{attribute 'GeneratedUsingTerminal: EK1100-0000-0018'}
{attribute addProperty BoxType "EK1100-0000-0018"}
{attribute addProperty Id "Beckhoff_EL66xxEK1122Beckhoff_EL66xxEK1122_DCCAD5BD273A_0001_EL6601_0000_0000EL6601_EEB2FEF410A_0002_EL6601_0000_0001EL6601_EEB2FEF410A_0003_EL6601_0000_0016EL6601_EEB2FEF410A_0004_EL6601_0000_0017EL6601_EEB2FEF410A_0005_EL6601_0000_0018EL6601_EEB2FEF410A_0006_EL6601_0000_0019EL6601_EEB2FEF410A_0007_EL6601_0000_0021EL6601_EEB2FEF410A_0008_EL6614_0000_0016EL6614_EEB2FEF410A_0009_EL6614_0000_0017EL6614_EEB2FEF410A_0010_EL6614_0000_0018EL6614_EEB2FEF410A_0011_EL6614_0000_0019EL6614_EEB2FEF410A_0012_EL6614_0000_0021EL6614_EEB2FEF410A_0013_EL6631_0000_0016EL6631_210A1A8D16A_0014_EL6631_0000_0017EL6631_210A1A8D16A_0015_EL6631_0000_0018EL6631_210A1A8D16A_0016_EL6631_0010_0016EL6631_210A1A8D16A_0017_EL6631_0010_0017EL6631_210A1A8D16A_0018_EL6631_0010_0018EL6631_210A1A8D16A_0019_EL6652_0000_0017EL6652_210A1A8D16A_0020_EL6652_0000_0018EL6652_210A1A8D16A_0021_EL6652_0010_0017EL6652_210A1A8D16A_0022_EL6652_0010_0018EL6652_210A1A8D16A_0023_EL6688_0000_0016EL6688_8DEED67724A_0024_EL6688_0000_0017EL6688_747A9CEE44A_0025_EL6688_0000_0018EL6688_747A9CEE44A_0026_EL6688_0000_0019EL6688_747A9CEE44A_0027_EL6688_0000_0020EL6688_747A9CEE44A_0028_EL6688_0000_0022EL6688_747A9CEE44A_0029_EL6690_0001_0000EL6690_FD149FC213A_0030_EL6690_0001_0016EL6690_FD149FC213A_0031_EL6690_0001_0017EL6690_FD149FC213A_0037_EL6692_0000_0016EL6692_F12D40B324A_0038_EL6692_0000_0017EL6692_F12D40B324A_0039_EL6692_0000_0018EL6692_F12D40B324A_0045_EL6695_0000_0001EL6695_258CDFB421A_0047_EL6695_0000_0002EL6695_258CDFB421A_0049_EL6695_0000_0003EL6695_258CDFB421A_0051_EL6695_0000_0004EL6695_258CDFB421A_0053_EL6695_0000_0005EL6695_258CDFB421A_0055_EL6695_0000_0006EL6695_258CDFB421"}
{attribute addProperty CRC "854866809"}
{attribute addProperty Size "1034"}
TYPE Beckhoff_EL66xx_32F43B79 EXTENDS EK1100_1FC0878B :
STRUCT
	{attribute addProperty Name "Beckhoff EL66xxEK1122"}
	{attribute addProperty PreviousPort "Beckhoff EL66xx : B"}
	Beckhoff_EL66xxEK1122 : Beckhoff_EL66xxEK1122_DCCAD5BD;
	{attribute addProperty Name "A_0001(EL6601-0000-0000)"}
	{attribute addProperty PreviousPort "Beckhoff EL66xxEK1122 : C"}
	A_0001_EL6601_0000_0000 : EL6601_EEB2FEF4;
	{attribute addProperty Name "A_0002(EL6601-0000-0001)"}
	{attribute addProperty PreviousPort "A_0001(EL6601-0000-0000) : B"}
	A_0002_EL6601_0000_0001 : EL6601_EEB2FEF4;
	{attribute addProperty Name "A_0003(EL6601-0000-0016)"}
	{attribute addProperty PreviousPort "A_0002(EL6601-0000-0001) : B"}
	A_0003_EL6601_0000_0016 : EL6601_EEB2FEF4;
	{attribute addProperty Name "A_0004(EL6601-0000-0017)"}
	{attribute addProperty PreviousPort "A_0003(EL6601-0000-0016) : B"}
	A_0004_EL6601_0000_0017 : EL6601_EEB2FEF4;
	{attribute addProperty Name "A_0005(EL6601-0000-0018)"}
	{attribute addProperty PreviousPort "A_0004(EL6601-0000-0017) : B"}
	A_0005_EL6601_0000_0018 : EL6601_EEB2FEF4;
	{attribute addProperty Name "A_0006(EL6601-0000-0019)"}
	{attribute addProperty PreviousPort "A_0005(EL6601-0000-0018) : B"}
	A_0006_EL6601_0000_0019 : EL6601_EEB2FEF4;
	{attribute addProperty Name "A_0007(EL6601-0000-0021)"}
	{attribute addProperty PreviousPort "A_0006(EL6601-0000-0019) : B"}
	A_0007_EL6601_0000_0021 : EL6601_EEB2FEF4;
	{attribute addProperty Name "A_0008(EL6614-0000-0016)"}
	{attribute addProperty PreviousPort "A_0007(EL6601-0000-0021) : B"}
	A_0008_EL6614_0000_0016 : EL6614_EEB2FEF4;
	{attribute addProperty Name "A_0009(EL6614-0000-0017)"}
	{attribute addProperty PreviousPort "A_0008(EL6614-0000-0016) : B"}
	A_0009_EL6614_0000_0017 : EL6614_EEB2FEF4;
	{attribute addProperty Name "A_0010(EL6614-0000-0018)"}
	{attribute addProperty PreviousPort "A_0009(EL6614-0000-0017) : B"}
	A_0010_EL6614_0000_0018 : EL6614_EEB2FEF4;
	{attribute addProperty Name "A_0011(EL6614-0000-0019)"}
	{attribute addProperty PreviousPort "A_0010(EL6614-0000-0018) : B"}
	A_0011_EL6614_0000_0019 : EL6614_EEB2FEF4;
	{attribute addProperty Name "A_0012(EL6614-0000-0021)"}
	{attribute addProperty PreviousPort "A_0011(EL6614-0000-0019) : B"}
	A_0012_EL6614_0000_0021 : EL6614_EEB2FEF4;
	{attribute addProperty Name "A_0013(EL6631-0000-0016)"}
	{attribute addProperty PreviousPort "A_0012(EL6614-0000-0021) : B"}
	A_0013_EL6631_0000_0016 : EL6631_210A1A8D;
	{attribute addProperty Name "A_0014(EL6631-0000-0017)"}
	{attribute addProperty PreviousPort "A_0013(EL6631-0000-0016) : B"}
	A_0014_EL6631_0000_0017 : EL6631_210A1A8D;
	{attribute addProperty Name "A_0015(EL6631-0000-0018)"}
	{attribute addProperty PreviousPort "A_0014(EL6631-0000-0017) : B"}
	A_0015_EL6631_0000_0018 : EL6631_210A1A8D;
	{attribute addProperty Name "A_0016(EL6631-0010-0016)"}
	{attribute addProperty PreviousPort "A_0015(EL6631-0000-0018) : B"}
	A_0016_EL6631_0010_0016 : EL6631_210A1A8D;
	{attribute addProperty Name "A_0017(EL6631-0010-0017)"}
	{attribute addProperty PreviousPort "A_0016(EL6631-0010-0016) : B"}
	A_0017_EL6631_0010_0017 : EL6631_210A1A8D;
	{attribute addProperty Name "A_0018(EL6631-0010-0018)"}
	{attribute addProperty PreviousPort "A_0017(EL6631-0010-0017) : B"}
	A_0018_EL6631_0010_0018 : EL6631_210A1A8D;
	{attribute addProperty Name "A_0019(EL6652-0000-0017)"}
	{attribute addProperty PreviousPort "A_0018(EL6631-0010-0018) : B"}
	A_0019_EL6652_0000_0017 : EL6652_210A1A8D;
	{attribute addProperty Name "A_0020(EL6652-0000-0018)"}
	{attribute addProperty PreviousPort "A_0019(EL6652-0000-0017) : B"}
	A_0020_EL6652_0000_0018 : EL6652_210A1A8D;
	{attribute addProperty Name "A_0021(EL6652-0010-0017)"}
	{attribute addProperty PreviousPort "A_0020(EL6652-0000-0018) : B"}
	A_0021_EL6652_0010_0017 : EL6652_210A1A8D;
	{attribute addProperty Name "A_0022(EL6652-0010-0018)"}
	{attribute addProperty PreviousPort "A_0021(EL6652-0010-0017) : B"}
	A_0022_EL6652_0010_0018 : EL6652_210A1A8D;
	{attribute addProperty Name "A_0023(EL6688-0000-0016)"}
	{attribute addProperty PreviousPort "A_0022(EL6652-0010-0018) : B"}
	A_0023_EL6688_0000_0016 : EL6688_8DEED677;
	{attribute addProperty Name "A_0024(EL6688-0000-0017)"}
	{attribute addProperty PreviousPort "A_0023(EL6688-0000-0016) : B"}
	A_0024_EL6688_0000_0017 : EL6688_747A9CEE;
	{attribute addProperty Name "A_0025(EL6688-0000-0018)"}
	{attribute addProperty PreviousPort "A_0024(EL6688-0000-0017) : B"}
	A_0025_EL6688_0000_0018 : EL6688_747A9CEE;
	{attribute addProperty Name "A_0026(EL6688-0000-0019)"}
	{attribute addProperty PreviousPort "A_0025(EL6688-0000-0018) : B"}
	A_0026_EL6688_0000_0019 : EL6688_747A9CEE;
	{attribute addProperty Name "A_0027(EL6688-0000-0020)"}
	{attribute addProperty PreviousPort "A_0026(EL6688-0000-0019) : B"}
	A_0027_EL6688_0000_0020 : EL6688_747A9CEE;
	{attribute addProperty Name "A_0028(EL6688-0000-0022)"}
	{attribute addProperty PreviousPort "A_0027(EL6688-0000-0020) : B"}
	A_0028_EL6688_0000_0022 : EL6688_747A9CEE;
	{attribute addProperty Name "A_0029(EL6690-0001-0000)"}
	{attribute addProperty PreviousPort "A_0028(EL6688-0000-0022) : B"}
	A_0029_EL6690_0001_0000 : EL6690_FD149FC2;
	{attribute addProperty Name "A_0030(EL6690-0001-0016)"}
	{attribute addProperty PreviousPort "A_0029(EL6690-0001-0000) : B"}
	A_0030_EL6690_0001_0016 : EL6690_FD149FC2;
	{attribute addProperty Name "A_0031(EL6690-0001-0017)"}
	{attribute addProperty PreviousPort "A_0030(EL6690-0001-0016) : B"}
	A_0031_EL6690_0001_0017 : EL6690_FD149FC2;
	{attribute addProperty Name "A_0037(EL6692-0000-0016)"}
	{attribute addProperty PreviousPort "A_0031(EL6690-0001-0017) : B"}
	A_0037_EL6692_0000_0016 : EL6692_F12D40B3;
	{attribute addProperty Name "A_0038(EL6692-0000-0017)"}
	{attribute addProperty PreviousPort "A_0037(EL6692-0000-0016) : B"}
	A_0038_EL6692_0000_0017 : EL6692_F12D40B3;
	{attribute addProperty Name "A_0039(EL6692-0000-0018)"}
	{attribute addProperty PreviousPort "A_0038(EL6692-0000-0017) : B"}
	A_0039_EL6692_0000_0018 : EL6692_F12D40B3;
	{attribute addProperty Name "A_0045(EL6695-0000-0001)"}
	{attribute addProperty PreviousPort "A_0039(EL6692-0000-0018) : B"}
	A_0045_EL6695_0000_0001 : EL6695_258CDFB4;
	{attribute addProperty Name "A_0047(EL6695-0000-0002)"}
	{attribute addProperty PreviousPort "A_0045(EL6695-0000-0001) : B"}
	A_0047_EL6695_0000_0002 : EL6695_258CDFB4;
	{attribute addProperty Name "A_0049(EL6695-0000-0003)"}
	{attribute addProperty PreviousPort "A_0047(EL6695-0000-0002) : B"}
	A_0049_EL6695_0000_0003 : EL6695_258CDFB4;
	{attribute addProperty Name "A_0051(EL6695-0000-0004)"}
	{attribute addProperty PreviousPort "A_0049(EL6695-0000-0003) : B"}
	A_0051_EL6695_0000_0004 : EL6695_258CDFB4;
	{attribute addProperty Name "A_0053(EL6695-0000-0005)"}
	{attribute addProperty PreviousPort "A_0051(EL6695-0000-0004) : B"}
	A_0053_EL6695_0000_0005 : EL6695_258CDFB4;
	{attribute addProperty Name "A_0055(EL6695-0000-0006)"}
	{attribute addProperty PreviousPort "A_0053(EL6695-0000-0005) : B"}
	A_0055_EL6695_0000_0006 : EL6695_258CDFB4;
END_STRUCT
END_TYPE

(* stored: Version 1.2.0.0, ProductVersion 3.1.4024.9
   DUT Beckhoff_EL66xx_32F43B79: Id {5ae504f9-b8e5-4ad8-879f-64964e694b69} *)
